Fanuc KAREL source: ka00131.KL

PROGRAM KA00131
%NOLOCKGROUP
VAR
SRC : ARRAY[2] OF BYTE
DST : ARRAY[2] OF BYTE
BEGIN
SRC[1]=2
DST[1]=SRC[1]
END KA00131
